// TIA Portal V15.1 export
// export: Created 2024-06-21T08:40:57.7774426Z, ExportSetting WithDefaults, DisplayName Totally Integrated Automation Portal, DisplayVersion V15.1 Update 5, DisplayName TIA Portal Openness, DisplayVersion V15.1 Update 5, DisplayName SINAMICS Startdrive Advanced, DisplayVersion V15.1, DisplayName G130, G150, S120, S150, SINAMICS MV, S210, DisplayVersion V15.1, DisplayName G110M, G120, G120C, G120D, G120P, DisplayVersion V15.1, DisplayName STEP 7 Professional, DisplayVersion V15.1 Update 5, DisplayName STEP 7 Safety, DisplayVersion V15.1, DisplayName WinCC Professional, DisplayVersion V15.1 Update 5, DisplayName SIMATIC Visualization Architect, DisplayVersion V15.1
FUNCTION_BLOCK "L2Alarm"   // FB1425, FBD
TITLE = L2Alarm
{ S7_Optimized_Access := 'FALSE' }
AUTHOR : VCC
FAMILY : AlarmHnd
NAME : 2Alarm
VERSION : 1.0
// ================================================================================
// This module is used everywhere two alarms shall be generated from one object.
// The alarm can be True only when the input Enable Alarm is also True.
// The alarm can be True only when the input Disable Alarm is False. When the 
// alarm is disable from HMI, a boolean output is available to inform the upper 
// level and do action in the Alarm summary.
// When the conditions to generate the alarm is disappear, a boolean output is 
// available to inform the upper level that the alarm can be reset.
// ================================================================================
// stored: AutoNumber false, IsIECCheckEnabled false, SetENOAutomatically False, UDAEnableTagReadback false
   VAR_INPUT
      I_Input1 { ExternalAccessible := 'False'; ExternalVisible := 'False'; ExternalWritable := 'False'} : Bool;   // Input signal 1 of the alarm
      I_AlarmClass1 { ExternalAccessible := 'False'; ExternalVisible := 'False'; ExternalWritable := 'False'} : Char;   // Alarm class -> A - B - C - D or E
      I_Input2 { ExternalAccessible := 'False'; ExternalVisible := 'False'; ExternalWritable := 'False'} : Bool;   // Input signal 2 of the alarm
      I_AlarmClass2 { ExternalAccessible := 'False'; ExternalVisible := 'False'; ExternalWritable := 'False'} : Char;   // Alarm class -> A - B - C - D or E
      I_EnableAlarm { ExternalAccessible := 'False'; ExternalVisible := 'False'; ExternalWritable := 'False'} : Bool := TRUE;   // Enable alarm from upper level
      I_AlarmResetPB { ExternalAccessible := 'False'; ExternalVisible := 'False'; ExternalWritable := 'False'} : Bool;   // Alarm reset pushbutton is activated
      I_Invisible { ExternalAccessible := 'False'; ExternalVisible := 'False'; ExternalWritable := 'False'} : Bool;   // Invisible
      C_NcAlarm { ExternalAccessible := 'False'; ExternalVisible := 'False'; ExternalWritable := 'False'} : Bool;   // Alarm contact NC
   END_VAR
   VAR_OUTPUT
      O_Alarm1 { ExternalAccessible := 'False'; ExternalVisible := 'False'; ExternalWritable := 'False'} : Bool;   // Alarm 1
      O_Alarm2 { ExternalAccessible := 'False'; ExternalVisible := 'False'; ExternalWritable := 'False'} : Bool;   // Alarm 2
      O_AlarmDisabled { ExternalAccessible := 'False'; ExternalVisible := 'False'; ExternalWritable := 'False'} : Bool;   // Alarm disabled from HMI
      O_AlarmABCondition { ExternalAccessible := 'False'; ExternalVisible := 'False'; ExternalWritable := 'False'} : Bool;   // Alarm AB condition
      H_IAnim1 { ExternalAccessible := 'False'; ExternalVisible := 'False'; ExternalWritable := 'False'} : Word;   // Icon Animation
      H_IAnim2 { ExternalAccessible := 'False'; ExternalVisible := 'False'; ExternalWritable := 'False'} : Word;   // Icon Animation
   END_VAR
   VAR DB_SPECIFIC
      H_In : Struct   // HMI
         DisableAlarm : Bool;   // Disable alarm from HMI
      END_STRUCT;
      H_Out : Struct   // HMI
         Anim1 : Word;   // HMI Animation of the object
         Anim2 : Word;   // HMI Animation of the object
         DBnr : Int;   // HMI Animation DB number
      END_STRUCT;
      Alarm1 { ExternalAccessible := 'False'; ExternalVisible := 'False'; ExternalWritable := 'False'} : Bool;   // Alarm 1
      AlarmClass1_A { ExternalAccessible := 'False'; ExternalVisible := 'False'; ExternalWritable := 'False'} : Bool;   // The alarm is from alarm class A
      AlarmClass1_B { ExternalAccessible := 'False'; ExternalVisible := 'False'; ExternalWritable := 'False'} : Bool;   // The alarm is from alarm class B
      AlarmClass1_C { ExternalAccessible := 'False'; ExternalVisible := 'False'; ExternalWritable := 'False'} : Bool;   // The alarm is from alarm class C
      AlarmClass1_D { ExternalAccessible := 'False'; ExternalVisible := 'False'; ExternalWritable := 'False'} : Bool;   // The alarm is from alarm class D
      AlarmClass1_E { ExternalAccessible := 'False'; ExternalVisible := 'False'; ExternalWritable := 'False'} : Bool;   // The alarm is from alarm class E
      AlarmCond1 { ExternalAccessible := 'False'; ExternalVisible := 'False'; ExternalWritable := 'False'} : Bool;   // Alarm condition 1
      Alarm2 { ExternalAccessible := 'False'; ExternalVisible := 'False'; ExternalWritable := 'False'} : Bool;   // Alarm 2
      AlarmClass2_A { ExternalAccessible := 'False'; ExternalVisible := 'False'; ExternalWritable := 'False'} : Bool;   // The alarm is from alarm class A
      AlarmClass2_B { ExternalAccessible := 'False'; ExternalVisible := 'False'; ExternalWritable := 'False'} : Bool;   // The alarm is from alarm class B
      AlarmClass2_C { ExternalAccessible := 'False'; ExternalVisible := 'False'; ExternalWritable := 'False'} : Bool;   // The alarm is from alarm class C
      AlarmClass2_D { ExternalAccessible := 'False'; ExternalVisible := 'False'; ExternalWritable := 'False'} : Bool;   // The alarm is from alarm class D
      AlarmClass2_E { ExternalAccessible := 'False'; ExternalVisible := 'False'; ExternalWritable := 'False'} : Bool;   // The alarm is from alarm class E
      AlarmCond2 { ExternalAccessible := 'False'; ExternalVisible := 'False'; ExternalWritable := 'False'} : Bool;   // Alarm condition 2
      DBnr { ExternalAccessible := 'False'; ExternalVisible := 'False'; ExternalWritable := 'False'} : Int;   // HMI DB number
   END_VAR
BEGIN

NETWORK
TITLE = **** 1 - Inputs **** DB number
// DB number
      L     DINO;
      T     #DBnr;

NETWORK
TITLE = **** 1 - Inputs **** Alarm class 1
// Alarm class
// Alarm class = E
      L     #I_AlarmClass1;
      L     'E';
      ==I;
      =     #AlarmClass1_E;

// Alarm class = D
      L     #I_AlarmClass1;
      L     'D';
      ==I;
      =     #AlarmClass1_D;

// Alarm class = C
      L     #I_AlarmClass1;
      L     'C';
      ==I;
      =     #AlarmClass1_C;

// Alarm class = B
      L     #I_AlarmClass1;
      L     'B';
      ==I;
      =     #AlarmClass1_B;

// Alarm class = A
      AN    #AlarmClass1_B;
      AN    #AlarmClass1_C;
      AN    #AlarmClass1_D;
      AN    #AlarmClass1_E;
      =     #AlarmClass1_A;


NETWORK
TITLE = **** 1 - Inputs **** Alarm class 2
// Alarm class
// Alarm class = E
      L     #I_AlarmClass2;
      L     'E';
      ==I;
      =     #AlarmClass2_E;

// Alarm class = D
      L     #I_AlarmClass2;
      L     'D';
      ==I;
      =     #AlarmClass2_D;

// Alarm class = C
      L     #I_AlarmClass2;
      L     'C';
      ==I;
      =     #AlarmClass2_C;

// Alarm class = B
      L     #I_AlarmClass2;
      L     'B';
      ==I;
      =     #AlarmClass2_B;

// Alarm class = A
      AN    #AlarmClass2_B;
      AN    #AlarmClass2_C;
      AN    #AlarmClass2_D;
      AN    #AlarmClass2_E;
      =     #AlarmClass2_A;


REGION Network 4: **** 2.2 - Alarms - Alarms Generation **** Alarm Condition 1
   // Condition of Alarm 1
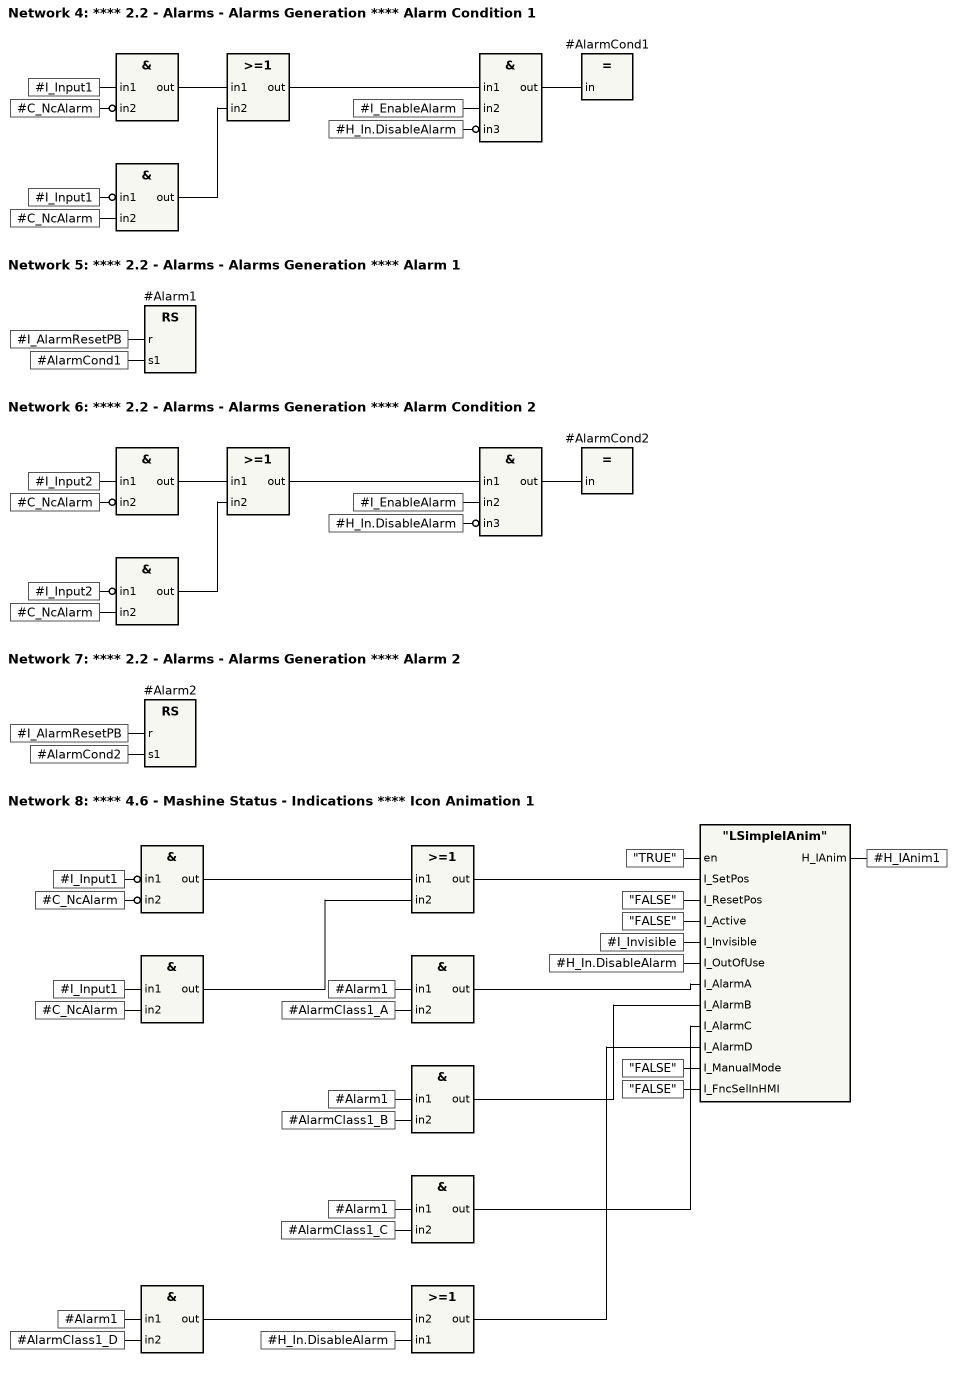
   #AlarmCond1 := ((#I_Input1 AND NOT #C_NcAlarm) OR (NOT #I_Input1 AND #C_NcAlarm)) AND #I_EnableAlarm AND NOT #H_In.DisableAlarm;
END_REGION

REGION Network 5: **** 2.2 - Alarms - Alarms Generation **** Alarm 1
   // Creation of Alarm 1
   IF #I_AlarmResetPB THEN
       #Alarm1 := FALSE;   // RS flip-flop
   END_IF;
   IF #AlarmCond1 THEN #Alarm1 := TRUE; END_IF;
END_REGION

REGION Network 6: **** 2.2 - Alarms - Alarms Generation **** Alarm Condition 2
   // Condition of Alarm 2
   #AlarmCond2 := ((#I_Input2 AND NOT #C_NcAlarm) OR (NOT #I_Input2 AND #C_NcAlarm)) AND #I_EnableAlarm AND NOT #H_In.DisableAlarm;
END_REGION

REGION Network 7: **** 2.2 - Alarms - Alarms Generation **** Alarm 2
   // Creation of Alarm 2
   IF #I_AlarmResetPB THEN
       #Alarm2 := FALSE;   // RS flip-flop
   END_IF;
   IF #AlarmCond2 THEN #Alarm2 := TRUE; END_IF;
END_REGION

REGION Network 8: **** 4.6 - Mashine Status - Indications **** Icon Animation 1
   // Icon Animation 1
   IF "TRUE" THEN
       "LSimpleIAnim"(I_SetPos := (NOT #I_Input1 AND NOT #C_NcAlarm) OR (#I_Input1 AND #C_NcAlarm),
                      I_ResetPos := "FALSE",
                      I_Active := "FALSE",
                      I_Invisible := #I_Invisible,
                      I_OutOfUse := #H_In.DisableAlarm,
                      I_AlarmA := #Alarm1 AND #AlarmClass1_A,
                      I_AlarmB := #Alarm1 AND #AlarmClass1_B,
                      I_AlarmC := #Alarm1 AND #AlarmClass1_C,
                      I_AlarmD := (#Alarm1 AND #AlarmClass1_D) OR #H_In.DisableAlarm,
                      I_ManualMode := "FALSE",
                      I_FncSelInHMI := "FALSE",
                      H_IAnim => #H_IAnim1);
   END_IF;
END_REGION

REGION Network 9: **** 4.6 - Mashine Status - Indications **** Icon Animation 2
   // Icon Animation 2
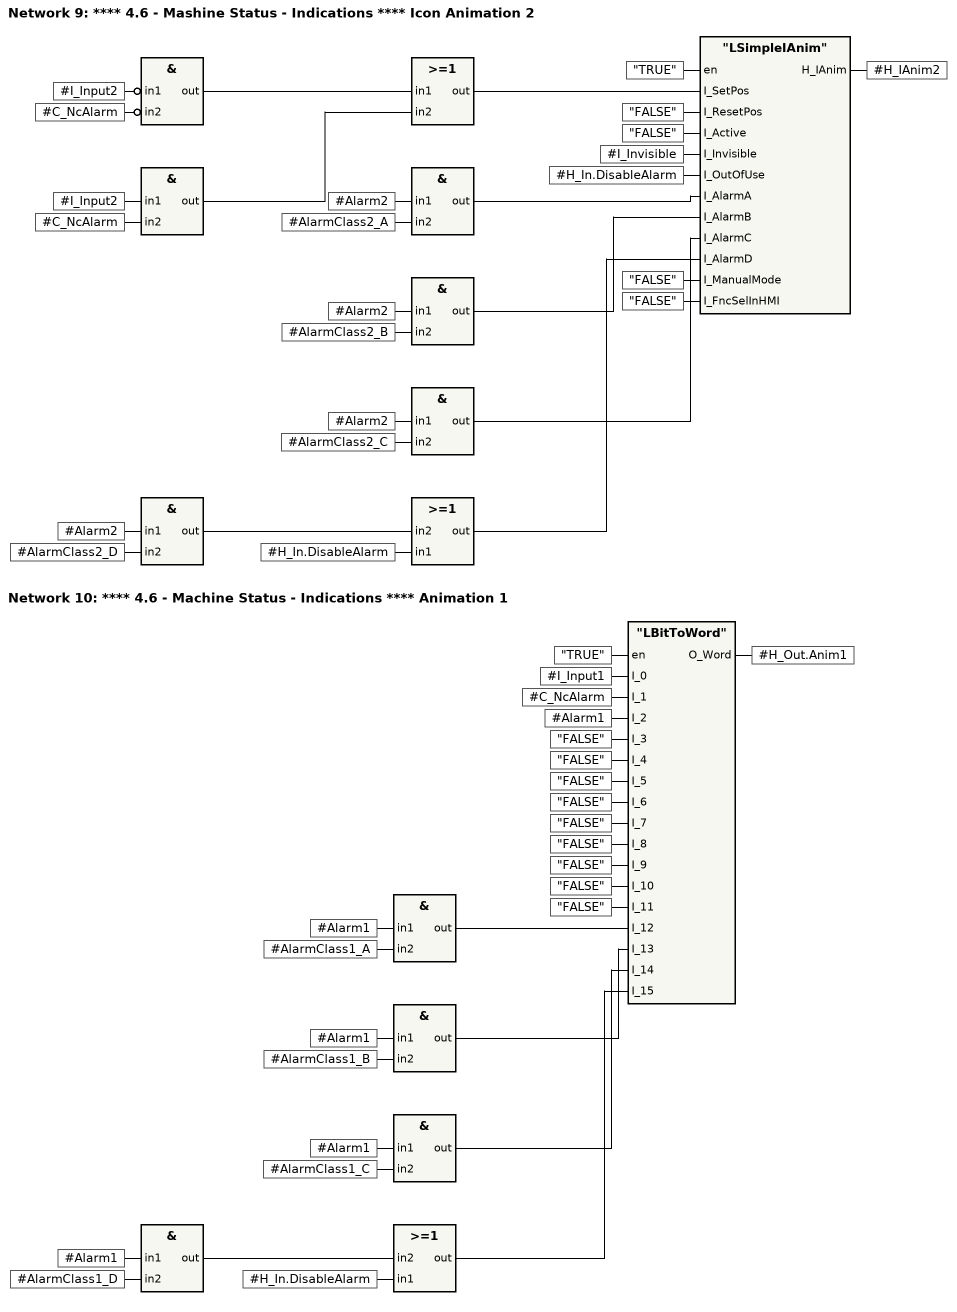
   IF "TRUE" THEN
       "LSimpleIAnim"(I_SetPos := (NOT #I_Input2 AND NOT #C_NcAlarm) OR (#I_Input2 AND #C_NcAlarm),
                      I_ResetPos := "FALSE",
                      I_Active := "FALSE",
                      I_Invisible := #I_Invisible,
                      I_OutOfUse := #H_In.DisableAlarm,
                      I_AlarmA := #Alarm2 AND #AlarmClass2_A,
                      I_AlarmB := #Alarm2 AND #AlarmClass2_B,
                      I_AlarmC := #Alarm2 AND #AlarmClass2_C,
                      I_AlarmD := (#Alarm2 AND #AlarmClass2_D) OR #H_In.DisableAlarm,
                      I_ManualMode := "FALSE",
                      I_FncSelInHMI := "FALSE",
                      H_IAnim => #H_IAnim2);
   END_IF;
END_REGION

REGION Network 10: **** 4.6 - Machine Status - Indications **** Animation 1
   // Animation 1
   IF "TRUE" THEN
       "LBitToWord"(I_0 := #I_Input1,
                    I_1 := #C_NcAlarm,
                    I_2 := #Alarm1,
                    I_3 := "FALSE",
                    I_4 := "FALSE",
                    I_5 := "FALSE",
                    I_6 := "FALSE",
                    I_7 := "FALSE",
                    I_8 := "FALSE",
                    I_9 := "FALSE",
                    I_10 := "FALSE",
                    I_11 := "FALSE",
                    I_12 := #Alarm1 AND #AlarmClass1_A,
                    I_13 := #Alarm1 AND #AlarmClass1_B,
                    I_14 := #Alarm1 AND #AlarmClass1_C,
                    I_15 := (#Alarm1 AND #AlarmClass1_D) OR #H_In.DisableAlarm,
                    O_Word => #H_Out.Anim1);
   END_IF;
END_REGION

REGION Network 11: **** 4.6 - Machine Status - Indications **** Animation 2
   // Animation 2
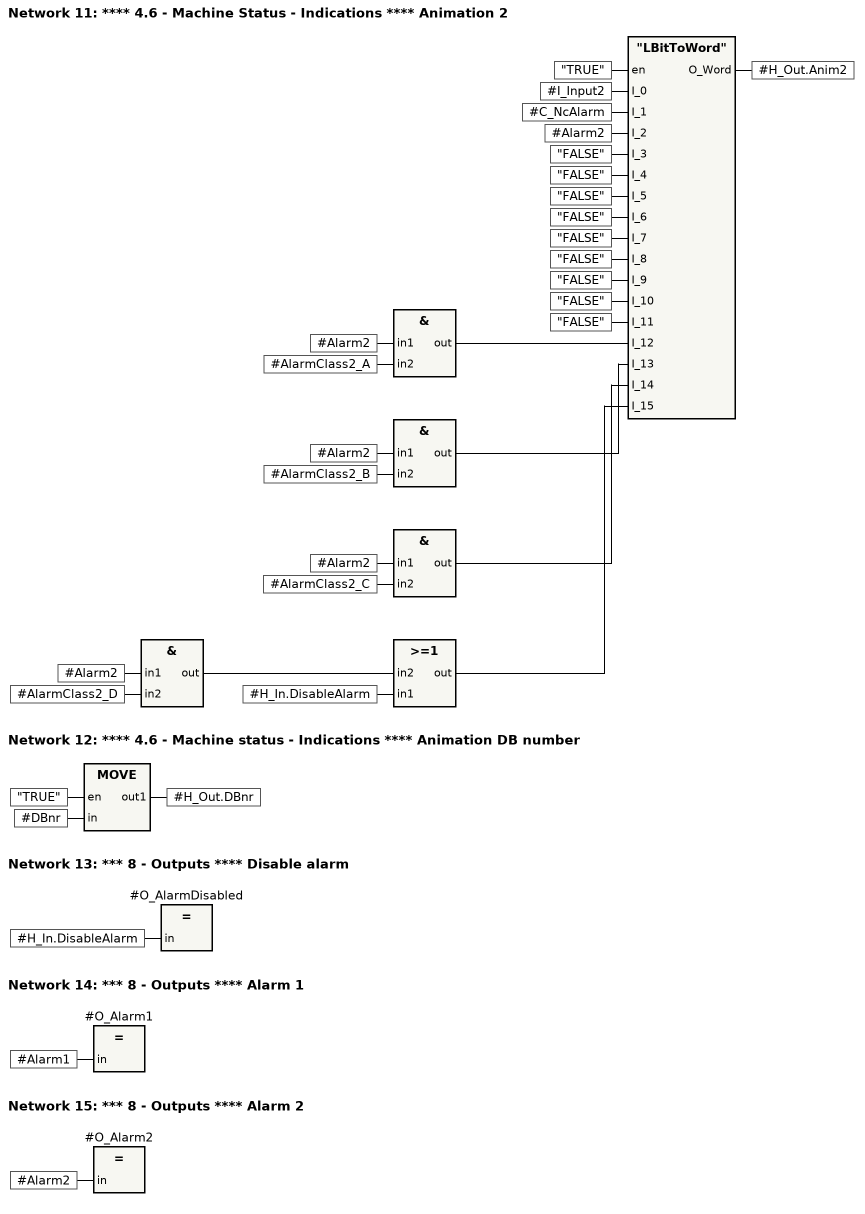
   IF "TRUE" THEN
       "LBitToWord"(I_0 := #I_Input2,
                    I_1 := #C_NcAlarm,
                    I_2 := #Alarm2,
                    I_3 := "FALSE",
                    I_4 := "FALSE",
                    I_5 := "FALSE",
                    I_6 := "FALSE",
                    I_7 := "FALSE",
                    I_8 := "FALSE",
                    I_9 := "FALSE",
                    I_10 := "FALSE",
                    I_11 := "FALSE",
                    I_12 := #Alarm2 AND #AlarmClass2_A,
                    I_13 := #Alarm2 AND #AlarmClass2_B,
                    I_14 := #Alarm2 AND #AlarmClass2_C,
                    I_15 := (#Alarm2 AND #AlarmClass2_D) OR #H_In.DisableAlarm,
                    O_Word => #H_Out.Anim2);
   END_IF;
END_REGION

REGION Network 12: **** 4.6 - Machine status - Indications **** Animation DB number
   IF "TRUE" THEN #H_Out.DBnr := #DBnr; END_IF;
END_REGION

REGION Network 13: *** 8 - Outputs **** Disable alarm
   // Alarm disabled from HMI
   #O_AlarmDisabled := #H_In.DisableAlarm;
END_REGION

REGION Network 14: *** 8 - Outputs **** Alarm 1
   // Output of the Alarm 1
   #O_Alarm1 := #Alarm1;
END_REGION

REGION Network 15: *** 8 - Outputs **** Alarm 2
   // Output of the Alarm 2
   #O_Alarm2 := #Alarm2;
END_REGION

REGION Network 16: **** 8 - Outputs **** Alarm AB Condition
   // Alarm AB condition
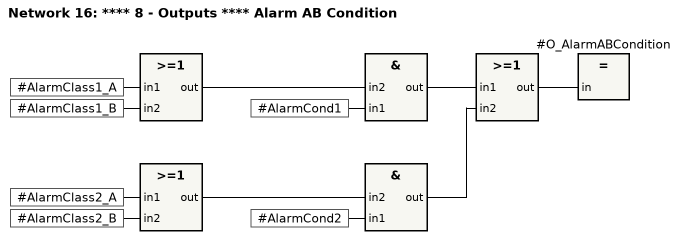
   #O_AlarmABCondition := ((#AlarmClass1_A OR #AlarmClass1_B) AND #AlarmCond1) OR ((#AlarmClass2_A OR #AlarmClass2_B) AND #AlarmCond2);
END_REGION
END_FUNCTION_BLOCK
